{attribute 'GeneratedUsingTerminal: AX8206-0100-0102-0102'}
{attribute addProperty BoxType "AX8206-0100-0102-0102"}
{attribute addProperty Id "Ch_B_AxisMain_InputsCh_B_AxisMain_Inputs_3D4AF9708Ch_B_AxisMain_OutputsCh_B_AxisMain_Outputs_526A47F82Ch_B_Interpolator_OutputsCh_B_Interpolator_Outputs_F819AE728Ch_B_PositionControl_InputsCh_B_PositionControl_Inputs_C884000A4"}
{attribute addProperty CRC "1686084108"}
{attribute addProperty Size "22"}
TYPE Ch_B_647F9A0C :
STRUCT
	{attribute addProperty Name "Ch_B_AxisMain_Inputs"}
	Ch_B_AxisMain_Inputs  : Ch_B_AxisMain_Inputs_3D4AF970;
	{attribute addProperty Name "Ch_B_AxisMain_Outputs"}
	Ch_B_AxisMain_Outputs  : Ch_B_AxisMain_Outputs_526A47F8;
	{attribute addProperty Name "Ch_B_Interpolator_Outputs"}
	Ch_B_Interpolator_Outputs  : Ch_B_Interpolator_Outputs_F819AE72;
	{attribute addProperty Name "Ch_B_PositionControl_Inputs"}
	Ch_B_PositionControl_Inputs  : Ch_B_PositionControl_Inputs_C884000A;
END_STRUCT
END_TYPE

(* stored: Version 1.2.0.0, ProductVersion 3.1.4024.9
   DUT Ch_B_647F9A0C: Id {b874f65a-18e2-4afa-8ffd-04781c8377ae} *)
